Staubli VAL3: PublicProg.pjx

--- PublicProg.pjx ---
Parameters version=s7.8.3 stackSize=5000 millimeterUnit=true
Program file=addBoolArray.pgx
Program file=addDirectory.pgx
Program file=addListItem.pgx
Program file=addMedscArray.pgx
Program file=addNumArray.pgx
Program file=addPointArray.pgx
Program file=addStrArray.pgx
Program file=addStrArray1.pgx
Program file=CompareTwoJoint.pgx
Program file=CompareTwoPoint.pgx
Program file=CopyStrArray.pgx
Program file=CutBlankLine.pgx
Program file=CutSpace.pgx
Program file=deletListItem.pgx
Program file=delJRsArray.pgx
Program file=delNumArray.pgx
Program file=delPointArray.pgx
Program file=delStrArray.pgx
Program file=delStrArray1.pgx
Program file=delToolArray.pgx
Program file=FileClose.pgx
Program file=FindStr.pgx
Program file=GetArrayIndex.pgx
Program file=JudgeSpace.pgx
Program file=SplitChar.pgx
Data file=PublicProg.dtx
Library alias=user path=Disk://userPage/USERPAGE.pjx

--- PublicProg.dtx ---
public mdesc mNomSpeed
public string sfliePath
string sContent

--- addBoolArray.pgx ---
public program addBoolArray(bool& x_In[], num x_nNum, bool& x_bRes)
  local num l_i
begin
  //建立指定数目的字符串数组
  //x_sStrIn:返回的新数组
  //x_nNum:数组个数
  //x_bRes:函数返回值
  x_bRes=false
  if x_nNum<1
    popUpMsg("新增点个数小于1")
    return
  endIf
  //取整
  x_nNum=roundDown(x_nNum)
  //删除原有的数组
  while size(x_In)>1
    delete(x_In[0])
  endWhile
  x_In[0]=false
  //插入新数据
  for l_i=1 to x_nNum-1
    insert(x_In[l_i])
  endFor
  x_bRes=true
end

--- addDirectory.pgx ---
public program addDirectory(bool& x_bRe, string x_sPath, string x_sDirName)
  local bool l_bool1
  local num l_i
begin
  //建立一个文件夹
  x_bRe=libList("Disk://",sContent)
  if !x_bRe
    return
  endIf

  if sContent[0]!=""
    x_bRe=$copy("Disk://"+sContent[0],x_sPath+"/"+x_sDirName)
    if !x_bRe
      return
    endIf
    x_bRe=libList(x_sPath+"/"+x_sDirName,sContent)
    if !x_bRe
      return
    endIf
    for l_i=0 to size(sContent)-1
      if sContent[l_i]!=""
        x_bRe=$delete(x_sPath+"/"+x_sDirName+"/"+sContent[l_i])
        if !x_bRe
          return
        endIf
      endIf
    endFor
  endIf
end

--- addListItem.pgx ---
public program addListItem(string& x_sName, string& x_sListName[], string x_sPrefix)
  local string l_sItemName
  local num l_nKey
  local num l_i
  local num l_nPos
begin
  //新建
  do
    call user:listframe("名称",10,5,20,1)
    call user:clear(11,6)
    gotoxy(15,6)
    l_nKey=get(l_sItemName)
    call JudgeSpace(l_i,l_sItemName)
    if l_nKey==270
      //输入为空,赋予一个值
      if l_sItemName==""
        l_i=0
        l_sItemName=x_sPrefix+toString("",l_i+1)
        while l_nPos!=-1
          call FindStr(l_sItemName,x_sListName,l_nPos)
          if l_nPos!=-1
            l_i=l_i+1
            l_sItemName=x_sPrefix+toString("",l_i+1)
          endIf
        endWhile
        x_sName=l_sItemName
      else
        call FindStr(l_sItemName,x_sListName,l_nPos)
        if l_nPos!=-1
          popUpMsg("重复，请重新输入")
          l_sItemName=""
        else
          x_sName=l_sItemName
          return
        endIf
      endIf
    endIf
    delay(0)
  until l_nKey==255
end

--- addMedscArray.pgx ---
public program addMedscArray(mdesc& x_In[], num x_nNum, bool& x_bRes)
  local num l_i
begin
  //建立指定数目的字符串数组
  //x_sStrIn:返回的新数组
  //x_nNum:数组个数
  //x_bRes:函数返回值
  x_bRes=false
  if x_nNum<1
    popUpMsg("新增点个数小于1")
    return
  endIf
  //取整
  x_nNum=roundDown(x_nNum)
  //删除原有的数组
  while size(x_In)>1
    delete(x_In[0])
  endWhile
  //插入新数据
  for l_i=1 to x_nNum-1
    insert(x_In[l_i])
  endFor
  x_bRes=true
end

--- addNumArray.pgx ---
public program addNumArray(num& x_In[], num x_nNum, bool& x_bRes)
  local num l_i
begin
  //建立指定数目的字符串数组
  //x_sStrIn:返回的新数组
  //x_nNum:数组个数
  //x_bRes:函数返回值
  x_bRes=false
  if x_nNum<1
    popUpMsg("新增点个数小于1")
    return
  endIf
  //取整
  x_nNum=roundDown(x_nNum)
  //删除原有的数组
  while size(x_In)>1
    delete(x_In[0])
  endWhile
  x_In[0]=-1
  //插入新数据
  for l_i=1 to x_nNum-1
   insert(x_In[l_i])
  endFor
  x_bRes=true
end

--- addPointArray.pgx ---
public program addPointArray(point& x_In[], num x_nNum, bool& x_bRes)
  local num l_i
begin
  //建立指定数目的字符串数组
  //x_sStrIn:返回的新数组
  //x_nNum:数组个数
  //x_bRes:函数返回值
  x_bRes=false
  if x_nNum<1
    popUpMsg("新增点个数小于1")
    return
  endIf
  //取整
  x_nNum=roundDown(x_nNum)
  //删除原有的数组
  while size(x_In)>1
    delete(x_In[0])
  endWhile
  //插入新数据
  for l_i=1 to x_nNum-1
    insert(x_In[l_i])
  endFor
  x_bRes=true
end

--- addStrArray.pgx ---
public program addStrArray(string& x_sStrIn[], num x_nNum, bool& x_bRes)
  local num l_i
begin
  //建立指定数目的字符串数组
  //x_sStrIn:返回的新数组
  //x_nNum:数组个数
  //x_bRes:函数返回值
  x_bRes=false
  if x_nNum<1
    popUpMsg("新增点个数小于1")
    return
  endIf
  //取整
  x_nNum=roundDown(x_nNum)
  //删除原有的数组
  while size(x_sStrIn)>1
    delete(x_sStrIn[0])
  endWhile
  x_sStrIn[0]=""
  //插入新数据
  for l_i=1 to x_nNum-1
    insert(x_sStrIn[l_i])
  endFor
  x_bRes=true
end

--- addStrArray1.pgx ---
public program addStrArray1(string& x_sStrIn[], num x_nPos, num x_nNum, bool& x_bRes)
  local num l_i
begin
  //建立指定数目的字符串数组
  //x_sStrIn:返回的新数组
  //x_nPos：指定位置
  //x_nNum:数组个数
  //x_bRes:函数返回值
  x_bRes=false
  if x_nNum<1
    popUpMsg("新增点个数小于1")
    return
  endIf
  if x_nPos<0
    x_nPos=0
  else
    if x_nPos>size(x_sStrIn)
      x_nPos=size(x_sStrIn)
    endIf
  endIf
  //取整
  x_nNum=roundDown(x_nNum)
   //插入新数据
  for l_i=x_nPos+1 to x_nPos+x_nNum
    insert(x_sStrIn[l_i])
  endFor
  x_bRes=true
end

--- CompareTwoJoint.pgx ---
public program CompareTwoJoint(joint x_jFirst, joint x_jSecond, bool& x_bSame, bool x_bIs6Axis)
  local joint l_jTolerance
begin
  //比较两个关节点是否相等
  x_bSame=false
  if x_bIs6Axis
    //六轴
    l_jTolerance={0.1,0.1,0.1,0.1}
    if abs(x_jFirst-x_jSecond)<l_jTolerance
        x_bSame=true
        return
    endIf
  else
    //四轴
    l_jTolerance={0.1,0.1,0.1,0.1,0.1,0.1}
    if abs(x_jFirst-x_jSecond)<l_jTolerance
        x_bSame=true
        return
    endIf
  endIf
end

--- CompareTwoPoint.pgx ---
public program CompareTwoPoint(point x_FirstPoint, point x_SecondPoint, bool& x_bSame)
begin
  //比较两个点是否相同
  x_bSame=false
  if distance(x_FirstPoint,x_SecondPoint)<0.5
    x_bSame=true
  endIf
end

--- CopyStrArray.pgx ---
public program CopyStrArray(string& x_sStrIn[], string& x_sStrOut[])
  local num i
begin
  //复制字符串数组
  while size(x_sStrOut)>1
    delete(x_sStrOut[0])
  endWhile
  x_sStrOut[0]=""
  while x_sStrIn[i]!=""
    x_sStrOut[i]=x_sStrIn[i]
  endWhile
end

--- CutBlankLine.pgx ---
public program CutBlankLine(num& x_nFileId, num& x_nLine, string& x_sLine)
begin
  do
    x_nLine=$fileGet(x_nFileId,x_sLine,1)
    if x_nLine<1
      return
    endIf
    call CutSpace(x_sLine,x_sLine)
    delay(0)
  until x_sLine!=""
end

--- CUTSPACE.pgx ---
public program CutSpace(string x_sStrIn, string& x_sStrOut)
begin
  //删除数据字符串中最后的空格
  if x_sStrIn!=""
    while right(x_sStrIn,1)==" "
      x_sStrIn=delete(x_sStrIn,1,len(x_sStrIn)-1)
    endWhile
  endIf
  x_sStrOut=x_sStrIn
  //
end

--- deletListItem.pgx ---
public program deletListItem(string& x_sList[], num x_nFirst, num& x_nSelect, bool& x_bListRefresh, bool& x_bRes)
  local string l_sYesNo[2]
  local num l_i
begin
  //F3:
  //x_nFirst:>=n(n>=1),按顺序保留的前n项
  //x_nFirst:0 不按顺序保留最后一项
  //x_nFirst:-1 全部删除,x_sList[0]=""
  x_bListRefresh=false
  x_bRes=false
  l_sYesNo[0]="是"
  l_sYesNo[1]="否"
  call user:questionDialog("是否删除该项?",l_sYesNo,l_i)
  if l_i==0 or l_i==1
    //
    x_nFirst=roundDown(x_nFirst)
    if x_nFirst==0
      if size(x_sList)==1
        popUpMsg("不能删除项!")
        return
      endIf
    endIf
    if size(x_sList)<=x_nFirst or x_nSelect<x_nFirst
      popUpMsg("不能删除项!")
      return
    endIf
    if size(x_sList)==1 and x_nFirst==-1
      x_sList=""
      x_bRes=true
      x_bListRefresh=true
      return
    endIf
    delete(x_sList[x_nSelect])
    x_nSelect=x_nSelect-1
    if x_nSelect<0
      x_nSelect=0
    endIf
    x_bListRefresh=true
    x_bRes=true
  endIf
end

--- delJRsArray.pgx ---
public program delJRsArray(jointRs& x_In[], num x_nNum)
  local num l_nSize
begin
  //删除字符串数组
  //x_sStrIn:返回的新数组
  //x_nNum:删除数组个数
  //取整
  x_nNum=roundDown(x_nNum)
  //
  l_nSize=size(x_In)
  if l_nSize<=1
    return
  endIf
  //
  if x_nNum>=l_nSize
    x_nNum=l_nSize-1
  endIf
  //
  while x_nNum>=1
    delete(x_In[0])
    x_nNum=x_nNum-1
  endWhile
end

--- delNumArray.pgx ---
public program delNumArray(num& x_sArrayIn[], num x_nNum)
  local num l_nSize
begin
  //删除字符串数组
  //x_sStrIn:返回的新数组
  //x_nNum:删除数组个数
  //取整
  x_nNum=roundDown(x_nNum)
  //
  l_nSize=size(x_sArrayIn)
  if l_nSize<=1
    x_sArrayIn=-1
    return
  endIf
  //
  if x_nNum>=l_nSize
    x_nNum=l_nSize-1
  endIf
  //
  while x_nNum>=1
    delete(x_sArrayIn[size(x_sArrayIn)-1])
    x_nNum=x_nNum-1
  endWhile
end

--- delPointArray.pgx ---
public program delPointArray(point& x_pIn[], num x_nNum)
  local num l_nSize
begin
  //删除字符串数组
  //x_sStrIn:返回的新数组
  //x_nNum:删除数组个数
  //取整
  x_nNum=roundDown(x_nNum)
  //
  l_nSize=size(x_pIn)
  if l_nSize<=1
    return
  endIf
  //
  if x_nNum>=l_nSize
    x_nNum=l_nSize-1
  endIf
  //
  while x_nNum>=1
    delete(x_pIn[size(x_pIn)-1])
    x_nNum=x_nNum-1
  endWhile
end

--- delStrArray.pgx ---
public program delStrArray(string& x_sStrIn[], num x_nNum)
  local num l_nSize
  local num l_i
begin
  //删除字符串数组
  //x_sStrIn:返回的新数组
  //x_nNum:删除数组个数
  //取整
  x_nNum=roundDown(x_nNum)
  //
  l_nSize=size(x_sStrIn)
  if l_nSize<=1
    x_sStrIn=""
    return
  endIf
  //
  if x_nNum>=l_nSize
    x_nNum=l_nSize-1
    x_sStrIn[0]=""
  endIf
  //

  while x_nNum>=1
    delete(x_sStrIn[size(x_sStrIn)-1])
    x_nNum=x_nNum-1
  endWhile

end

--- delStrArray1.pgx ---
public program delStrArray1(string& x_sStrIn[], num x_nPos, num x_nNum)
  local num l_nSize
  local num l_i
begin
  //删除字符串数组
  //x_sStrIn:返回的新数组
  //x_nPos：起始位置
  //x_nNum:删除数组个数
  //取整
  x_nNum=roundDown(x_nNum)
  if x_nNum<1
    return
  endIf
  if x_nNum>size(x_sStrIn)
    x_nNum=size(x_sStrIn)
  endIf

  //
  if x_nPos<0
    x_nPos=0
  else
    if x_nPos>size(x_sStrIn)-1
      x_nPos=size(x_sStrIn)-1
    endIf
  endIf
  //
  if size(x_sStrIn)<=1
    x_sStrIn=""
    return
  endIf
  //
  for l_i=x_nPos to min(size(x_sStrIn)-1,x_nPos+x_nNum-1)
    delete(x_sStrIn[size(x_sStrIn)-1])
  endFor
end

--- delToolArray.pgx ---
public program delToolArray(tool& x_In[], num x_nNum)
  local num l_nSize
begin
  //删除字符串数组
  //x_sStrIn:返回的新数组
  //x_nNum:删除数组个数
  //取整
  x_nNum=roundDown(x_nNum)
  //
  l_nSize=size(x_In)
  if l_nSize<=1
    return
  endIf
  //
  if x_nNum>=l_nSize
    x_nNum=l_nSize-1
  endIf
  //
  while x_nNum>=1
    delete(x_In[0])
    x_nNum=x_nNum-1
  endWhile
end

--- FileClose.pgx ---
public program FileClose()
  local num l_ni
begin

  $fileClose(0)
  $fileClose(1)
  $fileClose(2)
  $fileClose(3)
  $fileClose(4)
  $fileClose(5)
  $fileClose(6)
  $fileClose(7)
  $fileClose(8)
  $fileClose(9)
end

--- FINDSTR.pgx ---
public program FindStr(string x_sFindStr, string& x_sStrArray[], num& x_nPos)
  local num l_nSize
  local num i
begin
  //在x_sStrArray中查找x_sFindStr
  //x_nPos:位置
  //
  l_nSize=size(x_sStrArray)
  for  i=0 to l_nSize-1
    if x_sFindStr==x_sStrArray[i]
      x_nPos=i
      return
    endIf
  endFor
  x_nPos=-1
end

--- GetArrayIndex.pgx ---
public program GetArrayIndex(string& x_In[], string x_sFindStr, num x_nSelect, num& x_nIndex)
  local num l_i
begin
  //查找x_sFindStr在x_In中细分类别的索引值
  //x_nSelect:x_In中的第x_nSelect+1个元素
  //找到返回x_Index,否则返回-1
  //例如：x_In=[0，a],[1，a],[3,b],[4,a],[5,b],[6,b];x_nSelect=3
  //因为x_In由[0,a],[1,a],[4,a]和[3,b],[5,b],[6,b]
  //当x_nSelect=3时，对x_In为[3,b]，而该值在[b]值为第一个，故 x_nIndex=0；
  x_nIndex=-1
  if x_nSelect>size(x_In)
    x_nSelect=size(x_In)-1
  endIf
  for l_i=0 to x_nSelect
    if find(x_In[l_i],x_sFindStr)!=-1
      x_nIndex=x_nIndex+1
    endIf
  endFor
end

--- JudgeSpace.pgx ---
public program JudgeSpace(num& x_nRes, string x_sStrIn)
  local num l_i
begin
  //判断一个字符串是否是空格字符串
  //x_nRes=0:非空格字符串
  //x_nRes=1:空格字符串
  //x_nRes=2:空字符串
  x_nRes=0
  if x_sStrIn==""
    x_nRes=2
    return
  endIf
  for l_i=0 to len(x_sStrIn)-1
    if left(x_sStrIn,1)==" "
      x_sStrIn=right(x_sStrIn,len(x_sStrIn)-1)
    else
      return
    endIf
  endFor
  x_nRes=1
end

--- OpenFile.pgx ---
public program OpenFile(string x_sFile, bool& x_bRes)
begin
  //
  nFileHandle=$fileOpen(x_sFile,"w")
  if nFileHandle>=0 and nFileHandle<=9
    x_bRes=true
  else
    x_bRes=false
    logMsg("打开文件失败:"+x_sFile)
  endIf
end

--- SplitChar.pgx ---
public program SplitChar(num& x_nRes, string x_sStrIn, string x_sChar, string& x_sOut[])
  local string l_sBuff
  local num l_nIndex
  local num l_nLen
  local num l_nCharLen
  local num l_nStrIndex
begin
  //****************************************************************
  //***************************************************************
  //函数名称：SplitChar
  //用途：  用于解析字符
  //创建日期：
  //作者：
  //联系方式：
  //备注：
  //版本修改说明：
  //****************************************************************
  //*****************************************************************
  //1.参数定义
  l_sBuff=""
  l_nIndex=0
  l_nLen=0
  while size(x_sOut)>1
    delete(x_sOut[0])
  endWhile
  x_sOut[0]=""

  //2.条件判断
  if x_sStrIn=="" or x_sChar==""
    x_nRes=-1
    return
  endIf
  l_nCharLen=len(x_sChar)

  //3.分割字符串
  while find(x_sStrIn,x_sChar)>=0
    l_nStrIndex=find(x_sStrIn,x_sChar)
    l_nLen=l_nCharLen+l_nStrIndex
    x_sOut[l_nIndex]=left(x_sStrIn,l_nStrIndex)
    l_nIndex=l_nIndex+1
    insert(x_sOut[l_nIndex])
    x_sStrIn=delete(x_sStrIn,l_nLen,0)
  endWhile
  if x_sStrIn!=""
    x_sOut[l_nIndex]=x_sStrIn
  else
    delete(x_sOut[l_nIndex])
  endIf
  x_nRes=0
end
